Universal Robots URScript: 2-movel.script

def P2movel():
  set_standard_analog_input_domain(0, 1)
  set_standard_analog_input_domain(1, 1)
  set_tool_analog_input_domain(0, 1)
  set_tool_analog_input_domain(1, 1)
  set_analog_outputdomain(0, 0)
  set_analog_outputdomain(1, 0)
  set_tool_voltage(0)
  set_tcp(p[0.0,0.0,0.0,0.0,0.0,0.0])
  set_payload(0.0)
  set_gravity([0.0, 0.0, 9.82])
  while (True):
    $ 1 "机器人程序"
    $ 2 "MoveL"
    $ 3 "路点_1"
    movel([-1.5531271926045864, -1.5411282835497886, -2.2251433931393123, -0.9706436052226612, 1.5962951154371898, 0.01657278970905923], a=1.2, v=0.25)
    $ 4 "路点_2"
    movel([-1.5353943329175568, -0.9022793570722047, -2.5992265285302105, -1.2349536926524713, 1.5967259686141817, 0.03430619917457362], a=1.2, v=0.25)
    $ 5 "路点_3"
    movel([-0.6118263081418513, -0.8978483714273437, -2.608271528383848, -1.2000897153354249, 1.6056306953075028, 0.9582941238097733], a=1.2, v=0.25)
    $ 6 "路点_4"
    movel([-1.0649304904206653, -1.5410328949546814, -2.2296519999284996, -0.9514033687784353, 1.6048192376338637, 0.5049172533983802], a=1.2, v=0.25)
  end
end
